// SIMATIC S7-200 project (STEP 7-Micro/WIN), CPU 224 REL 01.21

ORGANIZATION_BLOCK 主:OB1
TITLE=【恒压供水控制系统（一）】
// 我实现了四个不同的恒压供水控制系统，这是第一个。
// 我的预想应用方式如下：
// 操作员通过按下系统启动按钮激活系统，随后可利用水泵启动按钮手动启动水泵1和水泵2，或依靠自动模式根据需求调节供水压力。系统通过压力传感器实时监测水压，并将数据存储在PID过程变量中。PID控制器根据压力设定值和实际压力计算出PID输出，通过变频器调整水泵速度以维持恒定压力。PID控制的运行在系统启动按钮按下、PID使能标志启用且水泵1运行时执行。
// 操作员可以通过压力设定调整按钮灵活调整压力设定值，以适应不同时段的用水需求。调整后的设定值和实际压力通过数显显示，让操作员能够直观监控系统状态。
// 系统内置了多重保护机制以应对故障。例如，若压力传感器故障检测到异常，系统会关闭水泵3，防止因压力数据不可靠导致的运行风险。同样，当水泵1故障、水泵2故障或水泵3故障任一触发时，系统会点亮对应的故障指示灯。若水泵1故障触发，点亮水泵1故障指示灯；若水泵2故障触发，点亮水泵2故障指示灯；若水泵3故障触发，点亮水泵3故障指示灯。当检测到水泵故障时，系统应禁用PID使能标志，以防止PID控制在故障条件下运行。
BEGIN
Network 1 // 通讯设置
//  
// 网络注释
//  
// 
LD     SM0.1
MOVB   16#49, SMB30
ATCH   INT_0:INT0, 8
MOVD   &VB999, VD10
MOVD   VD10, VD16
MOVW   +0, VW14
R      V100.0, 6
R      Q0.0, 2
S      V100.0, 1
ENI
Network 2 // 压力设定
// 
// 
LD     SM0.0
LPS
ITD    VW106, VD500
AW<>   VW106, VW512
S      M0.1, 1
LRD
A      M0.1
ITD    VW106, VD508
LRD
MOVW   VW106, VW512
LRD
A      I0.7
EU
A      V100.0
A      I0.0
AD<=   VD508, +1190
+D     +10, VD508
R      M0.1, 1
LRD
A      V100.6
EU
A      V100.0
A      I0.0
AD<=   VD508, +1190
+D     +10, VD508
R      M0.1, 1
LRD
A      I1.0
EU
A      V100.0
A      I0.0
AD>=   VD508, +10
-D     +10, VD508
R      M0.1, 1
LRD
A      V100.7
EU
A      V100.0
A      I0.0
AD>=   VD508, +10
-D     +10, VD508
R      M0.1, 1
LPP
DTI    VD508, VW109
DTR    VD508, VD504
MOVR   VD504, VD214
/R     5000.0, VD214
R      V100.6, 2
Network 3 // 模拟量处理
// 
// 
LD     SM0.0
MOVW   AIW0, VW602
-I     VW600, VW602
LDW>   VW602, +30
OW<    VW602, -30
ALD
MOVW   AIW0, VW600
Network 4
LD     SM0.0
CALL   数显:SBR0
CALL   恒压供水系统:SBR7
Network 5
LD     SM0.7
=      SM30.0
Network 6
LD     M0.0
TON    T33, +10
Network 7
LD     T33
AW>=   VW14, +7
AW=    VW1000, 16#5657
AW=    VW1005, 16#1003
AB=    VB1004, 1
CALL   SBR_1:SBR1
Network 8
LD     T33
AW>=   VW14, +7
AD=    VD1000, 16#52454144
AW=    VW1005, 16#1003
AB=    VB1004, 1
CALL   SBR_2:SBR2
Network 9
LD     T33
R      M0.0, 1
MOVW   +0, VW14
MOVD   VD10, VD16
END_ORGANIZATION_BLOCK

SUBROUTINE_BLOCK 数显:SBR0
TITLE= 
// 子程序注释
// 按 F1 获得帮助及举例程序
//  
BEGIN
Network 1 // 网络题目 (单行)
//  
// 网络注释
//  
// 
LD     SM0.1
S      M20.0, 1
Network 2
LD     M20.2
=      M20.1
Network 3
LD     C0
=      M20.2
R      M20.0, 1
Network 4
LD     M20.0
AN     C0
AN     M20.3
=      M20.3
Network 5
LD     M20.3
LD     C0
CTU    C0, +16
Network 6
LD     M20.1
S      M20.0, 1
Network 7
LD     SM0.0
LPS
AN     M20.2
=      Q0.6
LRD
AN     M20.3
=      Q0.7
LRD
AN     V2400.7
=      Q1.0
LPP
AN     V2600.7
=      Q1.1
Network 8
LDN    T51
MOVW   16#F9FF, VW2300
MOVW   16#FAF8, VW2302
MOVW   16#FBFF, VW2304
MOVW   16#FCFF, VW2306
Network 9
LD     SM0.1
MOVW   VW2300, VW2400
MOVD   &VB2300, VD4048
Network 10
LD     SM0.0
MOVD   &VB2306, VD4052
Network 11
LD     M20.3
SLW    VW2400, 1
Network 12
LD     M20.1
LPS
AD<    VD4048, VD4052
+D     +2, VD4048
MOVW   *VD4048, VW2400
MOVW   *VD4048, VW2450
LPP
AD>=   VD4048, VD4052
MOVD   &VB2298, VD4048
Network 13
LD     T51
LPS
AW>=   VW600, +6400
MOVW   VW600, VW250
-I     +6400, VW250
LRD
AW<    VW600, +6400
MOVW   +0, VW250
LRD
DTR    VD248, VD252
LRD
MOVR   VD252, VD256
/R     5.12, VD256
LRD
ROUND  VD256, VD260
LRD
DTI    VD260, VW264
LPP
MOVW   VW264, VW2350
IBCD   VW2350
Network 14
LD     T51
MOVW   VW2350, VW2352
ANDW   16#F000, VW2352
SWAP   VW2352
MOVW   VW2352, VW2354
SRW    VW2354, 4
MOVW   VW2354, VW2300
ORW    16#100, VW2300
AB=    VB2355, 0
AW>=   VW2350, +0
MOVW   16#10F, VW2300
Network 15
LD     T51
MOVW   VW2350, VW2356
ANDW   16#F00, VW2356
SWAP   VW2356
MOVW   VW2356, VW2302
ORW    16#2F0, VW2302
Network 16
LD     T51
MOVW   VW2350, VW2358
ANDW   16#F0, VW2358
MOVW   VW2358, VW2360
SRW    VW2360, 4
MOVW   VW2360, VW2304
ORW    16#300, VW2304
Network 17
LD     T51
MOVW   VW2350, VW2362
ANDW   16#F, VW2362
MOVW   VW2362, VW2306
ORW    16#400, VW2306
Network 18
LDN    SM0.1
TON    T51, +100
Network 19
LDN    T52
MOVW   16#F9FF, VW2500
MOVW   16#FAF8, VW2502
MOVW   16#FBFF, VW2504
MOVW   16#FCFF, VW2506
Network 20
LD     SM0.1
MOVW   VW2500, VW2600
MOVD   &VB2500, VD4056
Network 21
LD     SM0.0
MOVD   &VB2506, VD4060
Network 22
LD     M20.3
SLW    VW2600, 1
Network 23
LD     M20.1
LPS
AD<    VD4056, VD4060
+D     +2, VD4056
MOVW   *VD4056, VW2600
MOVW   *VD4056, VW2650
LPP
AD>=   VD4056, VD4060
MOVD   &VB2498, VD4056
Network 24
LD     T52
MOVW   VW109, VW2550
IBCD   VW2550
Network 25
LD     T52
MOVW   VW2550, VW2552
ANDW   16#F000, VW2552
SWAP   VW2552
MOVW   VW2552, VW2554
SRW    VW2554, 4
MOVW   VW2554, VW2500
ORW    16#100, VW2500
AB=    VB2555, 0
AW>=   VW2550, +0
MOVW   16#10F, VW2500
Network 26
LD     T52
MOVW   VW2550, VW2556
ANDW   16#F00, VW2556
SWAP   VW2556
MOVW   VW2556, VW2502
ORW    16#2F0, VW2502
Network 27
LD     T52
MOVW   VW2550, VW2558
ANDW   16#F0, VW2558
MOVW   VW2558, VW2560
SRW    VW2560, 4
MOVW   VW2560, VW2504
ORW    16#300, VW2504
Network 28
LD     T52
MOVW   VW2550, VW2562
ANDW   16#F, VW2562
MOVW   VW2562, VW2506
ORW    16#400, VW2506
Network 29
LDN    SM0.1
TON    T52, +100
END_SUBROUTINE_BLOCK

SUBROUTINE_BLOCK SBR_1:SBR1
TITLE=
BEGIN
Network 1
LD     SM0.0
MOVD   &VB100, VD20
ANDD   16#FF, VD999
+D     VD999, VD20
MOVB   VB1003, *VD20
END_SUBROUTINE_BLOCK

SUBROUTINE_BLOCK SBR_2:SBR2
TITLE=
BEGIN
Network 1
LD     SM0.0
LPS
A      I0.0
=      V104.7
LRD
A      I0.4
=      V104.4
LRD
A      I0.5
=      V104.5
LRD
A      I0.6
=      V104.6
LRD
A      Q0.0
=      V104.0
LRD
A      Q0.2
=      V105.0
LRD
A      Q0.3
=      V104.1
LRD
A      Q0.4
=      V104.2
LPP
A      Q0.5
=      V104.3
Network 2
LD     SM0.0
MOVD   16#52454144, VD96
MOVW   16#1003, VW150
MOVB   56, VB95
XMT    VB95, 0
END_SUBROUTINE_BLOCK

SUBROUTINE_BLOCK 恒压供水系统:SBR7
TITLE=
BEGIN
Network 1
LD     SM0.0
LPS
LD     I0.4
O      V100.3
ALD
A      Q0.0
=      Q0.3
LRD
LD     I0.5
O      V100.4
ALD
A      Q0.0
=      Q0.4
LRD
LD     I0.6
O      V100.5
ALD
A      Q0.0
=      Q0.5
LPP
AN     Q0.0
R      V100.3, 3
Network 2 // PID参数设定
// 
// 
LD     SM0.1
MOVR   0.9, VD222
MOVR   0.1, VD226
MOVR   0.3, VD230
MOVR   0.0, VD234
MOVB   9, VB115
MOVB   30, VB116
MOVB   0, VB117
S      V105.1, 3
Network 3 // INTOUCH画面上的PID参数的设定
// 
// 
LD     SM0.0
LPS
A      V105.1
MOVB   VB115, VB163
DTR    VD160, VD164
MOVR   VD164, VD222
/R     10.0, VD222
LRD
A      V105.2
MOVB   VB116, VB171
DTR    VD168, VD172
MOVR   VD172, VD230
/R     100.0, VD230
LPP
A      V105.3
MOVB   VB117, VB179
DTR    VD176, VD180
MOVR   VD180, VD234
/R     100.0, VD234
Network 4 // 水泵启动
// 
// 
LD     I0.1
O      V100.1
O      Q0.0
AN     I0.2
AN     V100.2
AN     Q0.2
=      Q0.0
=      Q0.1
Network 5
LDN    I0.3
=      Q0.2
Network 6
LD     SM0.0
LPS
AW<    VW600, +6400
MOVW   +6400, VW102
LRD
AW>=   VW600, +6400
MOVW   VW600, VW102
LPP
R      V100.1, 2
Network 7 // 过程变量的处理(实际压力)
// 
// 
LD     SM0.0
ITD    VW600, VD400
MOVD   VD400, VD404
-D     +6400, VD404
DTR    VD404, VD408
MOVR   VD408, VD210
/R     25600.0, VD210
Network 8
LD     SM0.0
LPS
AR<=   VD210, 0.0
MOVR   0.0, VD210
LPP
AR>=   VD210, 1.0
MOVR   1.0, VD210
Network 9
LD     I0.0
A      V100.0
A      Q0.0
PID    VB210, 0
Network 10 // 输出值的处理
// 
// 
LD     SM0.0
MOVR   VD218, VD424
*R     32000.0, VD424
ROUND  VD424, VD428
DTI    VD428, VW246
Network 11 // 手动时输出 的处理
// 
// 
LDN    I0.0
ON     V100.0
MOVW   +16000, AQW0
MOVB   25, VB108
Network 12
LD     I0.0
A      V100.0
MOVW   VW246, AQW0
MOVR   VD218, VD184
*R     50.0, VD184
ROUND  VD184, VD188
DTI    VD188, VW192
ITB    VW192, VB108
END_SUBROUTINE_BLOCK

INTERRUPT_BLOCK INT_0:INT0
TITLE= 
// 中断程序注释
// 按 F1 获得帮助及举例程序
//  
BEGIN
Network 1 // 网络题目 (单行)
//  
// 网络注释
//  
// 
LD     SM0.0
AW<=   VW14, +20
INCD   VD16
INCW   VW14
MOVB   SMB2, *VD16
=      M0.0
END_INTERRUPT_BLOCK
